// TIA Portal V16 export
Internal_Tag_BOOL :   ()

External_Tag_INT :   ()

Motor_Status_Text :   ()
